// TIA Portal V19 export
VAR_GLOBAL   // PLC tag table "U2Em2_Input"
   trayLiftingCylinderHomePositionDetectionU2Em2_2 AT %I174.1 : Bool;   // U2Em2_托盘顶升气缸原位检测2
   negativeLimitForCellJackingAndTransplantingU2Em2 AT %I175.6 : Bool;   // U2Em2_电池顶升移栽负限
   "palletScrewAnti-reverseDetectionU2Em2" AT %I42.3 : Bool;   // U2Em2_托盘螺杆防反检测
   positioningPinCylinderWorkingPositionDetectionU2Em2_2 AT %I43.6 : Bool;   // U2Em2_定位销气缸工作位检测2
   cellLiftingCylinderWorkingPositionDetectionU2Em2_1 AT %I43.0 : Bool;   // U2Em2_电池顶升气缸工作位检测1
   trayLiftingCylinderWorkingPositionDetectionU2Em2_2 AT %I174.0 : Bool;   // U2Em2_托盘顶升气缸工作位检测2
   positioningPinCylinderHomePositionDetectionU2Em2_1 AT %I43.5 : Bool;   // U2Em2_定位销气缸原位检测1
   positioningPinCylinderWorkingPositionDetectionU2Em2_1 AT %I43.4 : Bool;   // U2Em2_定位销气缸工作位检测1
   cellLiftingCylinderHomePositionDetectionU2Em2_2 AT %I43.3 : Bool;   // U2Em2_电池顶升气缸原位检测2
   originalForCellJackingAndTransplantingU2Em2 AT %I175.7 : Bool;   // U2Em2_电池顶升移栽原点
   cellLiftingCylinderHomePositionDetectionU2Em2_1 AT %I43.1 : Bool;   // U2Em2_电池顶升气缸原位检测1
   trayEntryDetectionU2Em2 AT %I42.0 : Bool;   // U2Em2_托盘进入检测
   trayInPlaceDetectionU2Em2 AT %I42.2 : Bool;   // U2Em2_托盘到位检测
   positioningPinCylinderHomePositionDetectionU2Em2_2 AT %I43.7 : Bool;   // U2Em2_定位销气缸原位检测2
   detectionBeforePalletPositioningU2Em2 AT %I42.4 : Bool;   // U2Em2_托盘定位前检测
   trayLiftingCylinderWorkingPositionDetectionU2Em2_1 AT %I42.6 : Bool;   // U2Em2_托盘顶升气缸工作位检测1
   positiveLimitForCellJackingAndTransplantingU2Em2 AT %I175.5 : Bool;   // U2Em2_电池顶升移栽正限
   detectionAfterTrayPositioningU2Em2 AT %I42.5 : Bool;   // U2Em2_托盘定位后检测
   cellLiftingCylinderWorkingPositionDetectionU2Em2_2 AT %I43.2 : Bool;   // U2Em2_电池顶升气缸工作位检测2
   trayLiftingCylinderHomePositionDetectionU2Em2_1 AT %I42.7 : Bool;   // U2Em2_托盘顶升气缸原位检测1
END_VAR
